Fanuc KAREL source: kt00495.KL

-- PROVISIONAL review KL for V1013-1; original PC SHA256 75b9583d576dd853749a3d2600d63e1925c0151082f1548d1bcbc25fe8c945da
-- Incomplete behavior may be omitted. Consult companion uncertainty JSON. Do not deploy.
PROGRAM KT00495
%NOLOCKGROUP
-- UNRESOLVED_DECL P1 type=000102
-- UNRESOLVED_DECL P2 type=000101
-- UNRESOLVED_DECL OUT type=000102
BEGIN
  -- UNRESOLVED_PC offsets 5-20; opcodes 2E,22,32,35
  -- UNRESOLVED_PC offsets 25-59; opcodes 49,7E,49,60,7E,4A
  -- UNRESOLVED_PC offsets 64-68; opcodes 7F
END KT00495
